Fanuc TP program (LS listing): GRP1_BLOWOFF.LS

/PROG  GRP1_BLOWOFF	  Macro
/ATTR
OWNER		= MNEDITOR;
COMMENT		= "Blow Gripper 1";
PROG_SIZE	= 572;
CREATE		= DATE 29-07-27  TIME 08:37:58;
MODIFIED	= DATE 29-07-27  TIME 08:37:58;
FILE_NAME	= ;
VERSION		= 0;
LINE_COUNT	= 19;
MEMORY_SIZE	= 1008;
PROTECT		= READ_WRITE;
TCD:  STACK_SIZE	= 1200,
      TASK_PRIORITY	= 50,
      TIME_SLICE	= 0,
      BUSY_LAMP_OFF	= 0,
      ABORT_REQUEST	= 0,
      PAUSE_REQUEST	= 0;
DEFAULT_GROUP	= *,*,*,*,*;
CONTROL_CODE	= 00000000 00000000;
/APPL
/MN
   1:  !******************************* ;
   2:  !COMPANY ;
   3:  !PROJECT 0000000 ;
   4:  !CUSTOMER Example Cell ;
   5:  ! ;
   6:  !Date: March 24, 2022 ;
   7:  ! ;
   8:  !Close (clamp) gripper 1 ;
   9:  !No error checking: ;
  10:  !******************************* ;
  11:  LBL[1:Begin] ;
  12:  !******************************* ;
  13:   ;
  14:  RO[1:Vacuum ON 1]=OFF ;
  15:  RO[2:Blowoff ON 1]=PULSE,5.0sec ;
  16:   ;
  17:  !Wait gripper close delay ;
  18:  //WAIT R[142] ;
  19:  CALL GRPSTAT1    ;
/POS
/END
